// TwinCAT 3 PLC project cream_module_shell
// ProgramVersion: 3.1.0.8
// libraries:
//   Tc2_Standard, * (Beckhoff Automation GmbH)
//   Tc2_System, * (Beckhoff Automation GmbH)
//   Tc3_Interfaces, * (Beckhoff Automation GmbH)
//   Tc3_Module, * (Beckhoff Automation GmbH)
//   Tc2_MC2,3.3.8.0,Beckhoff Automation GmbH
//   Tc2_TcpIp,3.3.2.0,Beckhoff Automation GmbH
//   Tc2_Utilities,3.3.7.0,Beckhoff Automation GmbH
// project tree:
//   DUTs/InternalDataTypes/ eMainState.TcDUT, eSubState.TcDUT
//   DUTs/Server DUTs/ DUT_MODE.TcDUT, DUT_PARAMETER_INPUT.TcDUT, DUT_PARAMETER_OUTPUT.TcDUT, DUT_SERVER_MODULE_INTERFACE.TcDUT, DUT_SERVER_MODULE_INTERFACE_INPUT.TcDUT, DUT_SERVER_MODULE_INTERFACE_OUTPUT.TcDUT, DUT_SERVER_PARAMETERINPUTARRAY.TcDUT, DUT_SERVER_PARAMETEROUTPUTARRAY.TcDUT, DUT_SERVER_SKILLINPUTARRAY.TcDUT, DUT_SERVER_SKILLOUTPUTARRAY.TcDUT, DUT_SERVER_SKILL_INPUT.TcDUT, DUT_SERVER_SKILL_OUTPUT.TcDUT, DUT_SERVER_STATEVALUEARRAY.TcDUT, DUT_STATEVALUES.TcDUT
//   DUTs/SimulationInterface/ MNG_APPLICATION_INPUTS_32BIT.TcDUT, MNG_APPLICATION_OUTPUTS_32BIT.TcDUT, MNG_DataArray.TcDUT, MNG_DatagramHeader.TcDUT, MNG_DatagramType.TcDUT, MNG_POSE6.TcDUT, MNG_RawDatagram.TcDUT, MNG_TRAFO.TcDUT, VEC3.TcDUT
//   GVLs/ GVL.TcGVL, MI5.TcGVL, MNG_GLOBALS.TcGVL, OPCConstants.TcGVL
//   / PlcTask.TcTTO, SimuTask.TcTTO
//   POUs/ FB_EmergencyStop.TcPOU, FB_Error.TcPOU, FB_Init.TcPOU, FB_MoveAbs.TcPOU, FB_MoveRel.TcPOU, FB_Ready.TcPOU, FB_Refill.TcPOU, FB_ResetAxis.TcPOU, FB_ResetSystem.TcPOU, FB_StorageLevel.TcPOU, FB_Timer.TcPOU, FB_LogFifo.TcPOU, MAIN.TcPOU, MAIN_simu.TcPOU, MNG_SIMULATION.TcPOU, MNG_UPDATEIOS.TcPOU
// real-time tasks:
//   TASK PlcTask: cycle T#10ms, priority 20, ADS port 350
//   TASK SimuTask: cycle T#10ms, priority 21, ADS port 351
// motion (NC):
//   TASK NC-Task 1 SAF: cycle T#2ms, priority 4, ADS port 501
//   TASK NC-Task 1 SVB: cycle T#10ms, priority 8, ADS port 511
//   AXIS Axis 1 (id 1)
//     OtherSettings: AllowMotionCmdToSlave=true
//     encoder EncType=8
//       EncPara: MaxCount=#x0036ee7f
//     drive DrvType=9
//       DrvPara: MaxCount=#xffffffff, DriveControlDWord=#x00030000
//         Analog: VeloScale=6
//         TimeComp: TaskDelayCycles=1
//     controller CtrType=1
//       CtrPara: PriorControlFactor=1
//         Observer: BandWidth=20
// I/O:
//   DEVICE Device 1 (EtherCAT), AmsNetId 5.27.156.253.2.1
//     Term 1 (EK1200) [EK1200-5000 EtherCAT Power supply (2A E-Bus)]
//       Term 2 (EL1804) [EL1804 4Ch. Dig. Input 24V, 3ms]
//       Term 3 (EL3162) [EL3162 2Ch. Ana. Input 0-10V]
//       Term 4 (EK1110) [EK1110 EtherCAT extension]
//     Drive 5 (IndraDrive MPB16/17) [IndraDrive MPB16/17]
//   DEVICE Device 3 (RT-Ethernet Protocol), AmsNetId 5.27.156.253.4.1
//   DEVICE Device 2 (NOV-DP-RAM)
// variable links:
//   NC-Task 1 SAF/Axes/Axis 1 <-> Device 1 (EtherCAT)/Drive 5 (IndraDrive MPB16/17)
//     Drive/Inputs/In/nDcOutputTime <-> InfoData/DcOutputShift
//     Drive/Inputs/In/nState1 <-> AT/Drive status word @bit 8
//     Drive/Inputs/In/nState2 <-> AT/Drive status word
//     Drive/Inputs/In/nState4 @bit 1 <-> WcState/InputToggle
//     Drive/Inputs/In/nState4 <-> WcState/WcState
//     Drive/Outputs/Out/nCtrl1 <-> MDT/Master control word @bit 8
//     Drive/Outputs/Out/nDataOut1 <-> MDT/Position command value
//     Enc/Inputs/In/nDataIn1 <-> AT/Position feedback value 1
//     Enc/Inputs/In/nDcInputTime <-> InfoData/DcInputShift
//     Enc/Inputs/In/nState4 @bit 1 <-> WcState/InputToggle
//     Enc/Inputs/In/nState4 <-> WcState/WcState
//   cream_module_shell/cream_module_shell Instance <-> Device 1 (EtherCAT)/Term 1 (EK1200)/Term 2 (EL1804)
//     PlcTask Inputs/GVL.init_sensor <-> Channel 4/Input
//   cream_module_shell/cream_module_shell Instance <-> Device 1 (EtherCAT)/Term 1 (EK1200)/Term 3 (EL3162)
//     PlcTask Inputs/GVL.iPositionSens <-> AI Standard Channel 1/Value
//   cream_module_shell/cream_module_shell Instance <-> NC-Task 1 SAF/Axes/Axis 1
//     PlcTask Inputs/GVL.axis.NcToPlc <-> Outputs/ToPlc
//     PlcTask Outputs/GVL.axis.PlcToNc <-> Inputs/FromPlc

CONFIGURATION cream_module_shell
    RESOURCE PLC ON TwinCAT3
        TASK PlcTask(INTERVAL := T#10ms, PRIORITY := 20);
        TASK SimuTask(INTERVAL := T#10ms, PRIORITY := 21);
        PROGRAM MAIN WITH PlcTask : MAIN;
        PROGRAM MAIN_simu WITH SimuTask : MAIN_simu;
    END_RESOURCE
END_CONFIGURATION

// ---- DUTs/InternalDataTypes/eMainState.TcDUT
TYPE eMainState :
(
	init			:= 0,
	ready			:= 10,
	output			:= 20,
	empty			:= 30,
	refill			:= 40,
	emergencyStop	:= 50,
	error			:= 60,
	resetSystem		:= 70
);
END_TYPE

// ---- DUTs/InternalDataTypes/eSubState.TcDUT
TYPE eSubState :
(
	step0 := 0,
	step1 := 10,
	step2 := 20,
	step3 := 30,
	step4 := 40,
	step5 := 50,
	step6 := 60,
	step7 := 70,
	step8 := 80,
	step9 := 90,
	step10 := 100,
	step11 := 110,
	step12 := 120,
	step13 := 130,
	step14 := 140,
	step15 := 150
);
END_TYPE

// ---- DUTs/Server DUTs/DUT_MODE.TcDUT
/// MODE to run (inside of MODULE_INTERFACE_INPUT)
TYPE DUT_MODE :
(
	///Initialitzation number mode
	Init := 0,
	///Automatic number mode
	Auto := 1,
	///Manual number mode
	Manual := 2,
	Reset := 3
);
END_TYPE

// ---- DUTs/Server DUTs/DUT_PARAMETER_INPUT.TcDUT
TYPE DUT_PARAMETER_INPUT :
STRUCT
	///Value of the parameter 
	Value: LREAL;
	///Possibility to a string value depending on the parameter
	StringValue: STRING(80);
END_STRUCT
END_TYPE

// ---- DUTs/Server DUTs/DUT_PARAMETER_OUTPUT.TcDUT
TYPE DUT_PARAMETER_OUTPUT :
STRUCT
	///Free to use = TRUE, busy to use =FALSE
	Dummy: BOOL := TRUE;
	///ID of the parameter
	ID: UINT;
	///Name of the parameter
	Name: STRING(80);
	///Unit of the parameter
	Unit: STRING(80);
	///Optional parameter
	Required: BOOL;
	///Default parameter to work
	Default: LREAL;
	///Minimum value of the parameter
	MinValue: LREAL;
	///Maximum value of the parameter
	MaxValue: LREAL;
END_STRUCT
END_TYPE

// ---- DUTs/Server DUTs/DUT_SERVER_MODULE_INTERFACE.TcDUT
/// MODULE INTERFACE INPUT AND OUTPUT 
TYPE DUT_SERVER_MODULE_INTERFACE :
STRUCT
	///Information that the module reads
	Input: DUT_SERVER_MODULE_INTERFACE_INPUT;
	///Information that the module write
	Output: DUT_SERVER_MODULE_INTERFACE_OUTPUT;
END_STRUCT
END_TYPE

// ---- DUTs/Server DUTs/DUT_SERVER_MODULE_INTERFACE_INPUT.TcDUT
TYPE DUT_SERVER_MODULE_INTERFACE_INPUT :
STRUCT
	///Mode to run (init,auto,manual,..)
	Mode: INT;
	///check if the modules is alive
	ConnectionTestInput: BOOL;
	///Modules get their position
	PositionInput : LREAL;
	///Update data= TRUE, No updatedata=FALSE
	Watchbit: BOOL;
	///Emergency stop
	EmergencyStop: BOOL;
	///Range of INPUT skills
	SkillInput: DUT_SERVER_SKILLINPUTARRAY;
END_STRUCT
END_TYPE

// ---- DUTs/Server DUTs/DUT_SERVER_MODULE_INTERFACE_OUTPUT.TcDUT
TYPE DUT_SERVER_MODULE_INTERFACE_OUTPUT :
STRUCT
	///Free to use = TRUE, busy to use =FALSE
	Dummy: BOOL := TRUE;
	///Individual name of the module
	Name: STRING(80);
	///Identification number of module
	ID: UINT;
	///IP address
	IP: STRING(80);
	///Show if the module is in Standby or not
	Idle: BOOL;
	///Show if the module is connected
	Connected: BOOL;
	///Feedback with conection test input
	ConnectionTestOutput: BOOL;
	///Show if the system has error when=TRUE
	Error: BOOL;
	///Identification number of the error
	ErrorID: UINT;
	///Description of the error
	ErrorDescription: STRING(80);
	///Description of the current task
	CurrentTaskDescription: STRING(80);
	///Position of the output
	PositionOutput: LREAL;
	/// Bool value of the Sensor
	PositionSensor: BOOL;
	///Range of OUTPUT skills
	SkillOutput: DUT_SERVER_SKILLOUTPUTARRAY;
	///Range of state values
	StateValue: DUT_SERVER_STATEVALUEARRAY;
END_STRUCT
END_TYPE

// ---- DUTs/Server DUTs/DUT_SERVER_PARAMETERINPUTARRAY.TcDUT
TYPE DUT_SERVER_PARAMETERINPUTARRAY :
STRUCT
	ParameterInput0: DUT_PARAMETER_INPUT;
	ParameterInput1: DUT_PARAMETER_INPUT;
	ParameterInput2: DUT_PARAMETER_INPUT;
	ParameterInput3: DUT_PARAMETER_INPUT;
	ParameterInput4: DUT_PARAMETER_INPUT;
	ParameterInput5: DUT_PARAMETER_INPUT;
END_STRUCT
END_TYPE

// ---- DUTs/Server DUTs/DUT_SERVER_PARAMETEROUTPUTARRAY.TcDUT
TYPE DUT_SERVER_PARAMETEROUTPUTARRAY :
STRUCT
	ParameterOutput0: DUT_PARAMETER_OUTPUT;
	ParameterOutput1: DUT_PARAMETER_OUTPUT;
	ParameterOutput2: DUT_PARAMETER_OUTPUT;
	ParameterOutput3: DUT_PARAMETER_OUTPUT;
	ParameterOutput4: DUT_PARAMETER_OUTPUT;
	ParameterOutput5: DUT_PARAMETER_OUTPUT;
END_STRUCT
END_TYPE

// ---- DUTs/Server DUTs/DUT_SERVER_SKILLINPUTARRAY.TcDUT
TYPE DUT_SERVER_SKILLINPUTARRAY :
STRUCT
	SkillInput0: DUT_SERVER_SKILL_INPUT;
	SkillInput1: DUT_SERVER_SKILL_INPUT;
	SkillInput2: DUT_SERVER_SKILL_INPUT;
	SkillInput3: DUT_SERVER_SKILL_INPUT;
	SkillInput4: DUT_SERVER_SKILL_INPUT;
	SkillInput5: DUT_SERVER_SKILL_INPUT;
	SkillInput6: DUT_SERVER_SKILL_INPUT;
	SkillInput7: DUT_SERVER_SKILL_INPUT;
	SkillInput8: DUT_SERVER_SKILL_INPUT;
	SkillInput9: DUT_SERVER_SKILL_INPUT;
	SkillInput10: DUT_SERVER_SKILL_INPUT;
	SkillInput11: DUT_SERVER_SKILL_INPUT;
	SkillInput12: DUT_SERVER_SKILL_INPUT;
	SkillInput13: DUT_SERVER_SKILL_INPUT;
	SkillInput14: DUT_SERVER_SKILL_INPUT;
	SkillInput15: DUT_SERVER_SKILL_INPUT;
END_STRUCT
END_TYPE

// ---- DUTs/Server DUTs/DUT_SERVER_SKILLOUTPUTARRAY.TcDUT
TYPE DUT_SERVER_SKILLOUTPUTARRAY :
STRUCT
	SkillOutput0: DUT_SERVER_SKILL_OUTPUT;
	SkillOutput1: DUT_SERVER_SKILL_OUTPUT;
	SkillOutput2: DUT_SERVER_SKILL_OUTPUT;
	SkillOutput3: DUT_SERVER_SKILL_OUTPUT;
	SkillOutput4: DUT_SERVER_SKILL_OUTPUT;
	SkillOutput5: DUT_SERVER_SKILL_OUTPUT;
	SkillOutput6: DUT_SERVER_SKILL_OUTPUT;
	SkillOutput7: DUT_SERVER_SKILL_OUTPUT;
	SkillOutput8: DUT_SERVER_SKILL_OUTPUT;
	SkillOutput9: DUT_SERVER_SKILL_OUTPUT;
	SkillOutput10: DUT_SERVER_SKILL_OUTPUT;
	SkillOutput11: DUT_SERVER_SKILL_OUTPUT;
	SkillOutput12: DUT_SERVER_SKILL_OUTPUT;
	SkillOutput13: DUT_SERVER_SKILL_OUTPUT;
	SkillOutput14: DUT_SERVER_SKILL_OUTPUT;
	SkillOutput15: DUT_SERVER_SKILL_OUTPUT;
END_STRUCT
END_TYPE

// ---- DUTs/Server DUTs/DUT_SERVER_SKILL_INPUT.TcDUT
TYPE DUT_SERVER_SKILL_INPUT :
STRUCT
	///Range of parameters
	ParameterInput: DUT_SERVER_PARAMETERINPUTARRAY;
	///Start process
	Execute: BOOL;
END_STRUCT
END_TYPE

// ---- DUTs/Server DUTs/DUT_SERVER_SKILL_OUTPUT.TcDUT
TYPE DUT_SERVER_SKILL_OUTPUT :
STRUCT
	///Free to use = TRUE, busy to use =FALSE
	Dummy: BOOL := TRUE;
	///Identification number of skill
	ID: UINT;
	///indentfication name of skill
	Name: STRING(80);
	///Skill activated
	Activated: BOOL;
	///Ready to do skill
	Ready: BOOL;
	///Skill in process
	Busy: BOOL;
	///Skill finish
	Done: BOOL;
	///Error in system
	Error: BOOL;
	///Range of parameters
	ParameterOutput: DUT_SERVER_PARAMETEROUTPUTARRAY;
END_STRUCT
END_TYPE

// ---- DUTs/Server DUTs/DUT_SERVER_STATEVALUEARRAY.TcDUT
TYPE DUT_SERVER_STATEVALUEARRAY :
STRUCT
	StateValue0: DUT_STATEVALUES;
	StateValue1: DUT_STATEVALUES;
	StateValue2: DUT_STATEVALUES;
	StateValue3: DUT_STATEVALUES;
	StateValue4: DUT_STATEVALUES;
	StateValue5: DUT_STATEVALUES;
	StateValue6: DUT_STATEVALUES;
	StateValue7: DUT_STATEVALUES;
	StateValue8: DUT_STATEVALUES;
	StateValue9: DUT_STATEVALUES;
	StateValue10: DUT_STATEVALUES;
END_STRUCT
END_TYPE

// ---- DUTs/Server DUTs/DUT_STATEVALUES.TcDUT
TYPE DUT_STATEVALUES :
STRUCT
	///Free to use = TRUE, busy to use =FALSE
	Dummy: BOOL := TRUE;
	///Value of the State
	Value: LREAL;
	///Name of the state
	Name: STRING(80);
	///Description of the state
	Description: STRING(80);
	///Unit of the state ()
	Unit: STRING(80);
END_STRUCT
END_TYPE

// ---- DUTs/SimulationInterface/MNG_APPLICATION_INPUTS_32BIT.TcDUT

TYPE MNG_APPLICATION_INPUTS_32BIT :
STRUCT
    NumSignals                     : INT     := 5         ;
    HallSensor1_00_IR : BOOL    := 0; (* ysics/Keksmodul/Keksmodul - relevant/HallSensor1?IR *)
    HallSensor2_00_IR : BOOL    := 0; (* ysics/Keksmodul/Keksmodul - relevant/HallSensor2?IR *)
    init_sensor_cookie_module_00_IR : BOOL    := 0; (* l/Keksmodul - relevant/init_sensor_cookie_module?IR *)
    kein_cookie_mehr_00_IR : BOOL    := 0; (* /Keksmodul/Keksmodul - relevant/kein_cookie_mehr?IR *)
    cookiebox_sensor_00_IR : BOOL    := 0; (* Physics://physics/Keksmodul/cookiebox_sensor?IR *)
END_STRUCT
END_TYPE

// ---- DUTs/SimulationInterface/MNG_APPLICATION_OUTPUTS_32BIT.TcDUT

TYPE MNG_APPLICATION_OUTPUTS_32BIT :
STRUCT
    NumSignals                     : INT     := 3         ;
    Disc_00_ACT_POS : REAL    := 0.0; (* ysics/Keksmodul/Keksmodul - relevant/Disc?KinActual *)
    A2014_09_12_Left_Predeterminado_00_ACT_POS : REAL    := 0.0; (* nt/Scissor/2014_09_12_Left_Predeterminado?KinActual *)
    A2014_09_12_Right_Predeterminado_00_ACT_POS : REAL    := 0.0; (* t/Scissor/2014_09_12_Right_Predeterminado?KinActual *)
END_STRUCT
END_TYPE

// ---- DUTs/SimulationInterface/MNG_DataArray.TcDUT
TYPE MNG_DataArray : ARRAY[1..MNG_BUFFER_SIZE] OF DWORD; (* user data of max. length *)
END_TYPE

// ---- DUTs/SimulationInterface/MNG_DatagramHeader.TcDUT
TYPE MNG_DatagramHeader :(* datagram header (4 byte aligned) *)
STRUCT
	(* Time when datagram has been created *)
	Counter 	: DWORD;
	(* Time when datagram has been sent *)
	SentTime 		: DWORD;
	(* Type of the datagram *)
	DatagramType 	: DWORD := MNG_UnknownDatagram;
	(* Byte count in the payload *)
	ByteCount 		: DWORD := 0;
END_STRUCT
END_TYPE

// ---- DUTs/SimulationInterface/MNG_DatagramType.TcDUT
TYPE MNG_DatagramType :
(
	(*Dead man datagram signalizing peer is alive *)
	MNG_DeadManDatagram := 0,
	(*Time tick synchonisation *)
	MNG_TimeTick,
	(*Time tick synchonisation *)
	MNG_TimeTickRequest,
	(*Initialization of the connection *)
	MNG_InitConnection,
	(*Reset simulation *)
	MNG_ResetSimulation,
	(*Rewind simulation *)
	MNG_RewindSimulation,
	(*Start simulation *)
	MNG_StartSimulation,
	(*Stop simulation *)
	MNG_StopSimulation,
	(*IO Config datagram *)
	MNG_IOConfig,
	(*Complete Raw IO Image *)
	MNG_RawIOImage,
	(*Complete Raw 32 Bit IO Image *)
	MNG_Raw32BitImage,
	(*Delta IO, only ios that have changed *)
	(* IODelta, *)
	(*Text datagram *)
	MNG_TextDatagram,
	(*Unknown Datagram (future updates of peer, not supported by this side) *)
	MNG_UnknownDatagram
);
END_TYPE

// ---- DUTs/SimulationInterface/MNG_POSE6.TcDUT
TYPE MNG_POSE6 :(* position and orientation as an euler based pose *)
STRUCT
	x, y, z, a, b, c : REAL;
END_STRUCT
END_TYPE

// ---- DUTs/SimulationInterface/MNG_RawDatagram.TcDUT
TYPE MNG_RawDatagram :(* binary TCP/IP datagram (4 byte aligned) *)
STRUCT
	Header	:  MNG_DatagramHeader;(* datagram header *)
	Payload	:  MNG_DataARRAY;
END_STRUCT
END_TYPE

// ---- DUTs/SimulationInterface/MNG_TRAFO.TcDUT
TYPE MNG_TRAFO :(* position and orientation as a 4x4 matrix *)
STRUCT
	baseX : VEC3; 
	fill0 : REAL;
	baseY : VEC3; 
	fill1 : REAL;
	baseZ : VEC3; 
	fill2 : REAL;
	origin : VEC3;
	fill3 : REAL;
END_STRUCT
END_TYPE

// ---- DUTs/SimulationInterface/VEC3.TcDUT
TYPE VEC3 :(* 3d position *)
STRUCT
	x, y, z : REAL;
END_STRUCT
END_TYPE

// ---- GVLs/GVL.TcGVL
VAR_GLOBAL
	pi : REAL := 3.14159;
																
	//<<Input Variables>>//
	iPositionSens	AT%I*	: INT;			// Position of extruder from sensor
	
	//OPC input Variables
	creamType				: INT;			// chocolate = 0, strawberry jam = 1, apricot jam = 2, cheese = 3
	optionalExtraCream		: INT;			// plenty = 0, normal = 1
	
	//<<Output Variables>>//
	oModulePosition			: LREAL;
	
	//<<Internal Variables>>//
	axis	 				: AXIS_REF;
	
	mainState 				: eMainState	:= eMainState.init;
	emptySubState			: eSubState 	:= eSubState.step0;	
	refillSubState			: eSubState		:= eSubState.step0;
	initSubState			: eSubState		:= eSubstate.step0;
	readySubState			: eSubState		:= eSubstate.step0;
	emergencySubState		: eSubState		:= eSubstate.step0;
	errorSubState			: eSubState		:= eSubstate.step0;
	resetSubState			: eSubState		:= eSubstate.step0;
	
	modulePositionInitialized	: BOOL := FALSE;	// is the module position initialized?
	firstRun					: bool := true;		// is this the first init? then wait for axis to get ready
	
	iMotorPosition			: LREAL;		//Position of extruder from motor encoder
	
	stepWidth				: LREAL;					//step width for motor to get optimal cream amount
	stepBackWidth			: LREAL;					//step width for motor to get optimal cream amount
	slowVel					: LREAL			:= 2.0;		// velocity for pressing cream out
	fastVel					: LREAL			:= 20.0;	// velocity for going back to full position
	fullPos					: LREAL			:= 89.0;	// Position where extruder is full
	emptyPos				: LREAL			:= 0.0;		// Position where extruder is empty

	//<<For Simulation>>//
	offset					: LREAL;
	infinitsimu				: BOOL;
	infinitsimu2			: BOOL;
	init_sensor		AT%I*	: BOOL;
	SensorPosition			: LREAL;
	
END_VAR

// ---- GVLs/MI5.TcGVL
VAR_GLOBAL
	//<<OPC-UA Module Interface>>//
	{attribute 'OPC.UA.DA' := '1'}
	Module2301 : DUT_SERVER_MODULE_INTERFACE;
	{attribute 'OPC.UA.DA' := '1'}
	mySkillID : INT := 1230;		//default: 1230 raspberry jam, 1240 for apple sauce, 1250 for apricot
	{attribute 'OPC.UA.DA' := '1'}
	reset : BOOL := false;
END_VAR

// ---- GVLs/MNG_GLOBALS.TcGVL

VAR_GLOBAL CONSTANT
	PLCPRJ_MAX_CONNECTIONS					: UDINT 	:= 5;   (* Max. number of server<->client connections *)
	PLCPRJ_SERVER_RESPONSE_TIMEOUT			: TIME 	:= T#10s;
	PLCPRJ_CLIENT_SEND_CYCLE_TIME			: TIME 	:= T#1ms;

	PLCPRJ_RECEIVER_POLLING_CYCLE_TIME		: TIME 	:= T#1ms;
	PLCPRJ_BUFFER_SIZE						: UDINT	:= 10000;   (* Max. internal fifo/receiver buffer size *)

	(* Some project specific error codes *)
	PLCPRJ_ERROR_RECEIVE_BUFFER_OVERFLOW	: UDINT := 16#8101; (* receive fifo/buffer overflow*)
	PLCPRJ_ERROR_SEND_BUFFER_OVERFLOW		: UDINT := 16#8102;	(* send fifo/buffer overflow *)
	PLCPRJ_ERROR_RESPONSE_TIMEOUT			: UDINT := 16#8103;	(* receive timeout error *)
	
	

	PLCPRJ_ERROR_INVALID_FRAME_FORMAT		: UDINT := 16#8104;	(* invalid frame format/data *)
	PLCPRJ_ERROR_INVALID_IO_FORMAT_RECEIVED : UDINT := 16#8105;	(* invalid io format/data *)
	PLCPRJ_ERROR_INTERNAL					: UDINT := 16#8105; (* internal error *)
	PLCPRJ_ERROR_RX_DATA_INCONSISTENT		: UDINT := 16#8106; (* rx data inconsistent *)
	
	PLCPRJ_ERROR_RECEIVE_TIMEOUT			: UDINT := 16#8107;
	PLCPRJ_ERROR_SENDFIFO_OVERFLOW			: UDINT := 16#8108; (* send fifo overflow error *)
	PLCPRJ_ERROR_RECFIFO_OVERFLOW			: UDINT := 16#8109; (* receive fifo overflow error *)
	
    MNG_BUFFER_SIZE						: DWORD := 32768;   (* Bytes: 131072; Max 128 KB of datagram payload data*)
	MNG_DatagramsFIFO_Size					: DWORD := 10;      (* Max 10 datagrams buffered before loss occurs *)
	MNG_EmptyDatagramHeader					: MNG_DatagramHeader;
	MNG_Application_NumInputs				: DWORD := 4;
	MNG_Application_NumOutputs				: DWORD := 4;

        (* PI should be defined by the system *)
        (* PI      : LREAL := 3.1415926535897932384626433832795; *)
        DEG2RAD : LREAL := 0.017453292519943295769236907684886;
        RAD2DEG : LREAL := 57.295779513082320876798154814105;
END_VAR

VAR_GLOBAL
        MNG_TIMESTAMP                                           : LREAL := 0;
END_VAR

// ---- GVLs/OPCConstants.TcGVL
VAR_GLOBAL CONSTANT
	///Maximum number of skillparameters
	ParameterCnt: INT := 5;
	///Maximum number of skills per Module
	SkillCnt: INT := 15;
	///Maximum number of Statevalues of one Module
	StateCnt: INT := 10;
	///Maximum number of modules
	ModuleCnt: INT := 10;
	///Maximum number of Tasks in Production List
	TaskCnt: INT := 30;
	///Maximum number  of offered recipes
	OfferCnt: INT := 5;
	///Maximum number of Orders in Queue
	OrderCnt: INT := 5;
	///Number of user set parameters per recipe
	UserParameterCnt: INT := 5;
	///Number of skills per task
	TaskSkillCnt: INT := 50;
END_VAR

// ---- POUs/MAIN.TcPOU
PROGRAM MAIN
VAR
	FBI_init			: FB_Init;			//FBI = function block instance
	FBI_refill			: FB_Refill;
	FBI_ready			: FB_Ready;
	FBI_emergencyStop 	: FB_EmergencyStop;
	FBI_error 			: FB_Error;
	FBI_storageLevel	: FB_StorageLevel;
	FBI_resetSystem		: FB_ResetSystem;  

	
	//jonas Interface variables:
	FBI_Timer			: TOF;
END_VAR

// @TODO measure position of slide against position sensor of XTS

//----------------------------------------- Error handling and emergency stop ------------------------------------------
axis.ReadStatus();

//reset system
IF (MI5.reset) THEN	
	GVL.mainState := eMainState.resetSystem;

//Emergency Stop Watchdog!	
ELSIF Module2301.Input.EmergencyStop THEN		
	GVL.mainState := eMainState.emergencyStop;

// error handling
ELSIF (axis.Status.Error) THEN					
	GVL.mainState := eMainState.error;
	
END_IF


//------------------------------------------------ OPC UA and module init --------------------------------------------------------------

//Connection Test
Module2301.Output.ConnectionTestOutput := Module2301.Input.ConnectionTestInput;
//positionsweitergabe an procvess tool
Module2301.Output.PositionOutput := Module2301.Input.PositionInput + 31;

//module positioning (by jf)
FBI_Timer();
IF GVL.init_sensor THEN
	Module2301.Output.PositionSensor := TRUE;
	FBI_Timer(IN := TRUE,PT := T#400MS);
	FBI_Timer(IN := FALSE,PT := T#400MS);
ELSE
	Module2301.Output.PositionSensor := FBI_Timer.Q;
END_IF


//----------------------------------------------- cream function process and parameter reading ----------------------------------------------------

// determine stepWidth from creamType
IF (MI5.mySkillID = 1230 OR MI5.mySkillID = 1250) THEN				// raspberry jam or apricot
	GVL.stepWidth := -3.5 - (Module2301.Input.SkillInput.SkillInput0.ParameterInput.ParameterInput0.Value / 100);
	GVL.stepBackWidth := 2;
ELSIF (MI5.mySkillID = 1240) THEN			// applesauce
	GVL.stepWidth := -4.5 - (Module2301.Input.SkillInput.SkillInput0.ParameterInput.ParameterInput0.Value / 100);
	GVL.stepBackWidth := 3;
END_IF


// get constantly the position of extruder
GVL.iMotorPosition := axis.NcToPlc.ActPos;

// update motor position for simulation
Module2301.Output.StateValue.StateValue2.Value := GVL.iMotorPosition;

//calculate storage level
FBI_storageLevel();


//----------------------------------------------- pseudo function block calls ----------------------------------------------------------------------

CASE GVL.mainState OF

	eMainState.init: //<<<<<<<<<<<<<<<<<<<<<<<<<<<<<<<<<<<<<<<<<<<<<<<<<<<<<<<<<<<<<<
		//init of state whereever the position of the disk is
		FBI_init();
	
	eMainState.ready: //<<<<<<<<<<<<<<<<<<<<<<<<<<<<<<<<<<<<<<<<<<<<<<<<<<<<<<<<<<<<<
		//cookie is on the clamps, waiting for putting it on the mover
		FBI_ready();
	
	eMainState.refill: //<<<<<<<<<<<<<<<<<<<<<<<<<<<<<<<<<<<<<<<<<<<<<<<<<<<<<<<<<<<<
		//cookie storage empty --> needs to be refilled
		FBI_refill();
		
	eMainState.emergencyStop: //<<<<<<<<<<<<<<<<<<<<<<<<<<<<<<<<<<<<<<<<<<<<<<<<<<<<<<<<<<<<
		// manually set emergency stop
		FBI_emergencyStop();
		
	eMainState.error: //<<<<<<<<<<<<<<<<<<<<<<<<<<<<<<<<<<<<<<<<<<<<<<<<<<<<<<<<<<<<
		// error state
		FBI_error();
		
	eMainState.resetSystem: //<<<<<<<<<<<<<<<<<<<<<<<<<<<<<<<<<<<<<<<<<<<<<<<<<<<<<<<<<<<<
		//error state
		FBI_resetSystem(); 
		
END_CASE

END_PROGRAM

// ---- POUs/FB_Init.TcPOU
FUNCTION_BLOCK FB_Init
VAR_INPUT
END_VAR
VAR_OUTPUT	
END_VAR
VAR
	resetAxis	: FB_ResetAxis;
	timer		: FB_Timer;
END_VAR

//@TODO: Determine the correct difference between sensor value and motorposition

//>>>OPCUA Init<<<
CASE initSubState OF	
			
step0:		// wait for everything to boot in first run
			IF (firstRun) THEN
				timer(iTime:=T#5S, execute := TRUE);
				IF(timer.done) THEN
					firstRun := FALSE;
				END_IF
			ELSE
				initSubState := step1;
			END_IF

step1:		//reset all substates
			emptySubState := step0;
			refillSubState := step0;
			readySubState := step0;
			emergencySubState := step0;
			errorSubState := step0;

			//>>>OPCUA Init<<<
			//>Module<
			Module2301.Output.ID := 2301;
			Module2301.Output.Name := 'Cream module Beckhoff';
			Module2301.Output.IP := '192.168.192.138';
			Module2301.Output.CurrentTaskDescription := 'Init process started: OPC UA';
			Module2301.Output.Dummy := FALSE;
			Module2301.Output.Idle := FALSE;
			Module2301.Output.Error := FALSE;
			Module2301.Output.ErrorDescription := '';
			Module2301.Output.ErrorID := 0;			
			
			//>Skill<:
			//Skill Cream
			Module2301.Output.SkillOutput.SkillOutput0.ID := mySkillID;
			Module2301.Output.SkillOutput.SkillOutput0.Activated := TRUE;
			Module2301.Output.SkillOutput.SkillOutput0.Busy := TRUE;
			Module2301.Output.SkillOutput.SkillOutput0.Done := FALSE;
			Module2301.Output.SkillOutput.SkillOutput0.Error := FALSE;
			Module2301.Output.SkillOutput.SkillOutput0.Ready := FALSE;
			Module2301.Output.SkillOutput.SkillOutput0.Dummy := FALSE;
			
			// publish maximum level of cream for HMI
			Module2301.Output.StateValue.StateValue1.Description := 'Maximum level of cream in injection.';
			Module2301.Output.StateValue.StateValue1.Dummy := FALSE;
			Module2301.Output.StateValue.StateValue1.Name := 'Max. Cream';
			Module2301.Output.StateValue.StateValue1.Unit := 'ml';
			Module2301.Output.StateValue.StateValue1.Value := 113;
			
			// publish motor position for simulation
			Module2301.Output.StateValue.StateValue2.Description := 'Motor Position.';
			Module2301.Output.StateValue.StateValue2.Dummy := FALSE;
			Module2301.Output.StateValue.StateValue2.Name := 'Motor Position';
			Module2301.Output.StateValue.StateValue2.Unit := 'mm';
			
			//initialize position input with value -1
			IF (NOT GVL.modulePositionInitialized)THEN
				Module2301.Input.PositionInput := -1;
				GVL.modulePositionInitialized := TRUE;
			END_IF
							
			resetAxis (execute := FALSE);
			
			IF (axis.Status.StandStill OR axis.Status.ErrorStop OR axis.Status.Disabled) THEN
				initSubState := step2;
			END_IF			

			
step2:		IF NOT resetAxis.done THEN
				// axreset
				resetAxis (execute := TRUE);
			ELSE
				initSubState := step3;
			END_IF
			
			
step3:		IF (iMotorPosition <=5) THEN
				mainState := eMainState.refill;
			ELSE
				mainState := eMainState.ready;
			END_IF
				initSubState := step0;
END_CASE

END_FUNCTION_BLOCK

// ---- POUs/FB_ResetAxis.TcPOU
FUNCTION_BLOCK FB_ResetAxis
VAR_INPUT
	execute: BOOL;
END_VAR
VAR_OUTPUT
	done : BOOL;
	busy : BOOL;
	error: BOOL;
END_VAR
VAR
	state			: INT := 0;
	fbreset			: Tc2_MC2.MC_Reset;
END_VAR

IF execute THEN
	CASE state OF
	
	0: 
		done := FALSE;
		fbreset(axis := axis, Execute := FALSE);
		state := 1;
		
	1:
		fbreset(
				Axis:= axis, 
				Execute:= TRUE, 
				Done=> , 
				Busy=> , 
				Error=> error, 
				ErrorID=> );
		IF fbreset.Done THEN
			state := 2;
		END_IF
		
	2:	
		execute := FALSE;
		done  := TRUE;
		state := 0;

	END_CASE
ELSE
	done := FALSE;
	state := 0;
END_IF

END_FUNCTION_BLOCK

// ---- POUs/FB_Timer.TcPOU
FUNCTION_BLOCK FB_Timer
VAR_INPUT
	iTime	: TIME;
	execute : Bool;
END_VAR
VAR_OUTPUT
	done	: BOOL;
END_VAR
VAR
	timer	: Tc2_Standard.TON;
	state	: INT := 0;
END_VAR

IF (execute) THEN
	
	CASE state OF
	
		0:	done := FALSE;
			timer(IN:= FALSE, PT:= iTime);
			timer(IN:= TRUE, PT:= iTime);
			state := 10;
	
		10:	timer();
			IF (timer.Q) THEN
				done := TRUE;
				state :=0;
			END_IF
	END_CASE

ELSE
	state := 0;
	done := FALSE;
END_IF

END_FUNCTION_BLOCK

// ---- POUs/FB_Refill.TcPOU
FUNCTION_BLOCK FB_Refill
VAR_INPUT
END_VAR
VAR_OUTPUT
END_VAR
VAR
	moveAbs : FB_MoveAbs;
END_VAR

CASE refillSubState OF

	step0:	//set OPC state variables
			Module2301.Output.SkillOutput.SkillOutput0.Busy := TRUE;
			Module2301.Output.SkillOutput.SkillOutput0.Done := FALSE;
			Module2301.Output.SkillOutput.SkillOutput0.Error := FALSE;
			Module2301.Output.SkillOutput.SkillOutput0.Ready := FALSE;
			
			//reset move functions
			moveAbs(execute := FALSE);
			
			refillSubState := step1; 
	
	step1:	//Move back to position with cream extruder beeing fully extended
			moveAbs(targetPos:= GVL.fullPos, targetVel:= GVL.fastVel, execute:= TRUE);
			IF (moveAbs.done) THEN
				refillSubState := step2; 
			END_IF
			

	step2:	//go in the right error state
			Module2301.Output.SkillOutput.SkillOutput0.Busy := FALSE;
			Module2301.Output.CurrentTaskDescription := 'Cream empty. Switching to refill mode.';
			Module2301.Output.ErrorID := 201;
			Module2301.Output.Error := TRUE;
			Module2301.Output.ErrorDescription := 'storage empty. please refill';
			refillSubState := step3;
			
	step3:	//wait for process tool to set the module in manual mode
			IF(Module2301.Input.Mode = DUT_MODE.Manual) THEN
				refillSubState := step4;
			END_IF
			
	step4:	//wait for process tool to set the module in init mode
			IF(Module2301.Input.Mode = DUT_MODE.Auto) THEN
				//reset error 
				Module2301.Output.Error := FALSE;
				Module2301.Output.ErrorDescription := '';
				Module2301.Output.ErrorID := 0;
				
				//change to ready state
				mainState := eMainState.ready;
				refillSubState := step0;
			END_IF
END_CASE

END_FUNCTION_BLOCK

// ---- POUs/FB_MoveAbs.TcPOU
FUNCTION_BLOCK FB_MoveAbs
VAR_INPUT
	targetPos		: LREAL;
	targetVel		: LREAL;
	execute			: BOOL := TRUE;
	
END_VAR

VAR_OUTPUT
	done 			: BOOL;
	moveAbs			: Tc2_MC2.MC_MoveAbsolute;
END_VAR

VAR
	state		: INT := -10;
	power		: Tc2_MC2.MC_Power;
END_VAR

//Comment here
IF (NOT execute) THEN
	state := -10;
	moveAbs	(Axis:= axis , Execute:= FALSE);
ELSE
	//Comment here
	power(
			Axis			:= axis , 
			Enable			:= TRUE , 
			Enable_Positive	:= TRUE , 
			Enable_Negative	:= TRUE , 
			BufferMode		:= Tc2_MC2.MC_BlendingNext
		);				
					
	CASE state OF 
		 
		-10:	//Comment here
				done := FALSE;
				IF (power.Status=TRUE AND power.Error=FALSE) THEN
					state := 0;
				END_IF
							
		0:		//Comment here
				moveAbs(Axis:= axis , Execute:= FALSE);
				state := 10;			
				
		10:		//Comment here
				IF (moveAbs.Done=FALSE) THEN
					moveAbs(Axis:= axis, Execute:= TRUE, Position:= targetPos, Velocity:=targetVel, BufferMode:= Tc2_MC2.MC_BlendingNext);
				ELSE 
					moveAbs(Axis:= axis, Execute:= FALSE);
					state := 20;
				END_IF
				
		20: 	//Comment here
				done 	:= TRUE;
				execute := false;
				state	:= -10;	
	END_CASE
END_IF

END_FUNCTION_BLOCK

// ---- POUs/FB_Ready.TcPOU
FUNCTION_BLOCK FB_Ready
VAR_INPUT
END_VAR
VAR_OUTPUT
END_VAR
VAR
	moveRel : FB_MoveRel;
END_VAR

CASE readySubState OF

step0:	moveRel(execute := false);
		IF (NOT (Module2301.Input.PositionInput = -1)) THEN
			readySubState := step1;
		END_IF

step1:	Module2301.Output.SkillOutput.SkillOutput0.Busy := FALSE;
		Module2301.Output.SkillOutput.SkillOutput0.Done := FALSE;
		Module2301.Output.SkillOutput.SkillOutput0.Error := FALSE;
		Module2301.Output.SkillOutput.SkillOutput0.Ready := TRUE;
		
		//wait for execute command
		IF(Module2301.Input.SkillInput.SkillInput0.Execute) THEN
		//order received
			Module2301.Output.SkillOutput.SkillOutput0.Ready := FALSE;
			Module2301.Output.SkillOutput.SkillOutput0.Busy := TRUE;
			readySubState := step2;
		END_IF
		
step2:	//@TODO: How much has the Bosch motor got to move to eject sufficient amount of cream?
		moveRel(targetDis:= GVL.stepWidth, targetVel:= GVL.slowVel, execute:= TRUE);
		IF (moveRel.done) THEN
			readySubState := step3; 
		END_IF
		
step3:	//@TODO: How much has the Bosch motor got to move to eject sufficient amount of cream?
		moveRel(targetDis:= GVL.stepBackWidth, targetVel:= GVL.slowVel, execute:= TRUE);
		IF (moveRel.done) THEN
			Module2301.Output.SkillOutput.SkillOutput0.Busy := FALSE;
			Module2301.Output.SkillOutput.SkillOutput0.Done := TRUE;
			readySubState := step4; 
		END_IF
		
step4:	// Test if distance sensor checks a position where the cream dispenser has to be empty
		IF (NOT Module2301.Input.SkillInput.SkillInput0.Execute) THEN
			IF (iMotorPosition <=5) THEN
				mainState := eMainState.refill;
			ELSE
				readySubState := step0;
			END_IF
		END_IF

END_CASE

END_FUNCTION_BLOCK

// ---- POUs/FB_MoveRel.TcPOU
FUNCTION_BLOCK FB_MoveRel
VAR_INPUT
	targetDis		: LREAL;
	targetVel		: LREAL;
	execute			: BOOL := TRUE;
	
END_VAR

VAR_OUTPUT
	done 			: BOOL;
	moveRel			: Tc2_MC2.MC_MoveRelative;
END_VAR

VAR
	state		: INT := -10;
	power		: Tc2_MC2.MC_Power;
END_VAR

//Comment here
IF (NOT execute) THEN
	state := -10;
	moveRel	(Axis:= axis , Execute:= FALSE);
ELSE
	//Comment here
	power(
			Axis			:= axis , 
			Enable			:= TRUE , 
			Enable_Positive	:= TRUE , 
			Enable_Negative	:= TRUE , 
			BufferMode		:= Tc2_MC2.MC_BlendingNext
		);				
					
	CASE state OF 
		 
		-10:	//Comment here
				done := FALSE;
				IF (power.Status=TRUE AND power.Error=FALSE) THEN
					state := 0;
				END_IF
							
		0:		//Comment here
				moveRel(Axis:= axis , Execute:= FALSE);
				state := 10;			
				
		10:		//Comment here
				IF (moveRel.Done=FALSE) THEN
					moveRel(Axis:= axis, Execute:= TRUE, Distance:= targetDis, Velocity:=targetVel, BufferMode:= Tc2_MC2.MC_BlendingNext);
				ELSE 
					moveRel(Axis:= axis, Execute:= FALSE);
					state := 20;
				END_IF
				
		20: 	//Comment here
				done 	:= TRUE;
				execute := false;
				state	:= -10;	
	END_CASE
END_IF

END_FUNCTION_BLOCK

// ---- POUs/FB_EmergencyStop.TcPOU
FUNCTION_BLOCK FB_EmergencyStop
VAR_INPUT
END_VAR
VAR_OUTPUT
END_VAR
VAR
END_VAR

CASE emergencySubState OF

	step0:	Module2301.Output.SkillOutput.SkillOutput0.Busy := FALSE;
			Module2301.Output.SkillOutput.SkillOutput0.Done := FALSE;
			Module2301.Output.SkillOutput.SkillOutput0.Dummy := FALSE;
			Module2301.Output.SkillOutput.SkillOutput0.Error := TRUE;
			Module2301.Output.SkillOutput.SkillOutput0.Ready := FALSE;
			
			//change in the right error state
			Module2301.Output.ErrorID := 302;
			Module2301.Output.CurrentTaskDescription := 'Emergency stop';
			Module2301.Output.Error := TRUE;
			Module2301.Output.ErrorDescription := 'Emergency stop. please solve problem';
			
			//wait for process tool to set the module in manual mode
			IF(Module2301.Input.Mode = DUT_MODE.Manual) THEN
				emergencySubState := step1;
			END_IF
			
	step1:	//wait for process tool to set the module in init mode
			IF(Module2301.Input.Mode = DUT_MODE.Auto) THEN
				//reset error 
				Module2301.Output.Error := FALSE;
				Module2301.Output.ErrorDescription := '';
				Module2301.Output.ErrorID := 0;

				//change to init state
				initSubState := step0;
				mainState := eMainState.init;
				emergencySubState := step0;
			END_IF
END_CASE

END_FUNCTION_BLOCK

// ---- POUs/FB_Error.TcPOU
FUNCTION_BLOCK FB_Error
VAR_INPUT
END_VAR
VAR_OUTPUT
END_VAR
VAR
	resetAxis			: FB_ResetAxis;
END_VAR

//@TODO: implement all possible errors

CASE errorSubState OF

	step0:	Module2301.Output.SkillOutput.SkillOutput0.Busy := FALSE;
			Module2301.Output.SkillOutput.SkillOutput0.Done := FALSE;
			Module2301.Output.SkillOutput.SkillOutput0.Dummy := FALSE;
			Module2301.Output.SkillOutput.SkillOutput0.Error := TRUE;
			Module2301.Output.SkillOutput.SkillOutput0.Ready := FALSE;
			
			// Error: axis got stuck
			IF (axis.Status.ErrorID = 17744) THEN
				Module2301.Output.ErrorDescription := 'Axis got stuck. Please clear module.';
				Module2301.Output.ErrorID := 301;
				errorSubState := step1;
			END_IF
			
			IF (Module2301.Output.ErrorID = 0) THEN
				Module2301.Output.ErrorDescription := 'Unknown Error.';
				Module2301.Output.ErrorID := 399;
				errorSubState := step1;
			END_IF
			
			//change in the right error state
			Module2301.Output.CurrentTaskDescription := 'Axis Error';
			Module2301.Output.Error := TRUE;
			
	step1:	//wait for process tool to set the module in manual mode
			IF(Module2301.Input.Mode = DUT_MODE.Manual) THEN
				resetAxis(execute:= FALSE);
				errorSubState := step2;
			END_IF
			
	step2:	IF NOT resetAxis.done THEN
				// axreset
				resetAxis (execute := TRUE);
			ELSE			
				errorSubState := step3;
			END_IF
			
	step3:	//wait for process tool to set the module in init mode
			IF(Module2301.Input.Mode = DUT_MODE.Auto) THEN
				//reset error 
				Module2301.Output.Error := FALSE;
				Module2301.Output.ErrorDescription := '';
				Module2301.Output.ErrorID := 0;
				
				//change to init state
				initSubState := step0;
				errorSubState := step0;
				mainState := eMainState.init;				
			END_IF
END_CASE

END_FUNCTION_BLOCK

// ---- POUs/FB_StorageLevel.TcPOU
FUNCTION_BLOCK FB_StorageLevel
VAR_INPUT
END_VAR
VAR_OUTPUT
END_VAR
VAR
	calculatedCream		: LREAL;
	remainingCream		: LREAL;		// in ml, is calculated by motor position
END_VAR

//Comment here	
IF (GVL.iPositionSens > 11090) THEN
	remainingCream := 0;
// configuration for all cookies (not as acurate)
ELSE
	calculatedCream := (11110 - GVL.iPositionSens)/86;
	remainingCream := REAL_TO_INT(calculatedCream);
END_IF

Module2301.Output.StateValue.StateValue0.Description := 'Remaining cream in the module.';
Module2301.Output.StateValue.StateValue0.Dummy := FALSE;
Module2301.Output.StateValue.StateValue0.Name := 'Remaining Cream';
Module2301.Output.StateValue.StateValue0.Unit := 'ml';
Module2301.Output.StateValue.StateValue0.Value := remainingCream;

END_FUNCTION_BLOCK

// ---- POUs/FB_ResetSystem.TcPOU
FUNCTION_BLOCK FB_ResetSystem
VAR_INPUT
END_VAR
VAR_OUTPUT
END_VAR
VAR
	resetAxis : FB_ResetAxis;
END_VAR

CASE GVL.resetSubState OF

step0:	resetAxis (execute := FALSE);

		Module2301.Output.SkillOutput.SkillOutput0.Busy := TRUE;
		Module2301.Output.SkillOutput.SkillOutput0.Done := TRUE;
		Module2301.Output.SkillOutput.SkillOutput0.Error := TRUE;
		Module2301.Output.SkillOutput.SkillOutput0.Ready := TRUE;
		
		GVL.resetSubState := step1;
		
step1:	IF NOT resetAxis.done THEN
		// axreset
		resetAxis (execute := TRUE);
		ELSE
			GVL.resetSubState := step2;
		END_IF
		
step2:	// reset substates
		GVL.emptySubState := step0;
		GVL.refillSubState := step0;
		GVL.initSubState := step0;
		GVL.readySubState := step0;
		GVL.emergencySubState := step0;
		GVL.errorSubState := step0;
		GVL.resetSubState := step0;
		
		MI5.reset := FALSE;
		GVL.mainState := eMainState.init;		
		
END_CASE

END_FUNCTION_BLOCK

// ---- POUs/MAIN_simu.TcPOU
PROGRAM MAIN_simu
VAR
    simIO 		: MNG_Simulation;
	outputs    	: MNG_Application_Outputs_32Bit;
    inputs     	: MNG_Application_Inputs_32Bit;
    ioUpdater  	: MNG_UpdateIOs                	:= (sRemoteHost := '192.168.175.222', nRemotePort := 5110);
	a 			: LREAL							:= 5.00;
    bEnable   	: BOOL                         	:= TRUE;
END_VAR

// Update IOs with simulation
//simIO(bEnable := TRUE);

// Application code follows here:
(*
IF GVL.infinitsimu THEN
	outputs.Disc_00_ACT_POS := (REAL_TO_INT(GVL.SensorPosition -180 + GVL.axis.NcToPlc.ModuloActPos))MOD 360;
ELSE
	IF GVL.infinitsimu2 THEN
		outputs.Disc_00_ACT_POS := (REAL_TO_INT(GVL.SensorPosition + GVL.axis.NcToPlc.ModuloActPos))MOD 360;
	ELSE
		outputs.Disc_00_ACT_POS := GVL.axis.NcToPlc.ModuloActPos;
	END_IF	
END_IF

storageLevel.full := inputs.kein_cookie_mehr_00_IR;

outputs.A2014_09_12_Right_Predeterminado_00_ACT_POS := ABS(SIN(((GVL.axis.NcToPlc.ActPos*pi)/180)))*(-7);
outputs.A2014_09_12_Left_Predeterminado_00_ACT_POS := ABS(SIN(((GVL.axis.NcToPlc.ActPos*pi)/180)))*(7);

GVL.iCookieInOutput := inputs.cookiebox_sensor_00_IR;
GVL.iDiskAtStorage := inputs.HallSensor1_00_IR;
GVL.iDiskAtRamp := inputs.HallSensor2_00_IR;

GVL.init_sensor := inputs.init_sensor_cookie_module_00_IR;

ioUpdater(Outputs := outputs, Inputs => inputs, bEnable := bEnable); 
*)
//outputs.Keksquelle_00_ReleaseTime := 60;
//outputs.Keksquelle_00_AlwaysOn := TRUE;

END_PROGRAM

// ---- POUs/MNG_SIMULATION.TcPOU
FUNCTION_BLOCK MNG_Simulation
VAR_INPUT
    bEnable    : BOOL                          := FALSE;
    outputs    : MNG_Application_Outputs_32Bit         ;
END_VAR
VAR_OUTPUT
    inputs     : MNG_Application_Inputs_32Bit          ;
END_VAR
VAR
    ioUpdater  : MNG_UpdateIOs                 := (sRemoteHost := '192.168.175.222', nRemotePort := 5110);
    fbCloseAll : FB_SocketCloseAll;
    bCloseAll  : BOOL := TRUE;
END_VAR

(* @END_DECLARATION := '0'                                                    *)
IF bCloseAll THEN (*On PLC reset or program download close all old (opened) connections *)
    bCloseAll := FALSE;
    fbCloseAll( bExecute:= TRUE );
ELSE
    fbCloseAll( bExecute:= FALSE );
END_IF

IF NOT fbCloseAll.bBusy THEN

    (* ------------------------------------- trigger data exchange ----------------------------------------------------------------------------*)
    ioUpdater(Outputs := outputs, Inputs => inputs, bEnable := bEnable);

END_IF

END_FUNCTION_BLOCK

// ---- POUs/MNG_UPDATEIOS.TcPOU
FUNCTION_BLOCK MNG_UpdateIOs
(* This function block implements simple TCP/IP client protocol.              *)
(* The max. size of binary tx/rx data has to be <= PLCPRJ_BUFFER_SIZE         *)
VAR_IN_OUT
    Outputs : MNG_Application_Outputs_32Bit;    (* Tx user data *)
END_VAR

VAR_INPUT
    bDbg        : BOOL                         := FALSE               ; (* TRUE => Enable debug output, FALSE => Disable debug output *)
    sRemoteHost : STRING(15)                   := '127.0.0.1'         ; (* IP address of remote server *)	
    nRemotePort : UDINT                        := 5000                ; (* Remote server port *)
    bEnable     : BOOL                         := FALSE               ; (* TRUE => Enable/connect, FALSE => Disable/disconnect *)
    tReconnect  : TIME                         := T#5s                ;
END_VAR

VAR_OUTPUT
    errors      : FB_LogFifo                                          ; (* Error message fifo *)
    Inputs      : MNG_Application_Inputs_32Bit                        ; (* Rx user data *)
    eState      : E_SocketConnectionState      := eSOCKET_DISCONNECTED; (* TCP/IP connection state *)
END_VAR

VAR
    counter          : DWORD                        := 0                   ;
    fbConnect        : FB_ClientServerConnection    := (tReconnect := T#5s); (* Create/release TCP/IP connection *)
    fbSend           : FB_SocketSend                                       ; (* Send TCP/IP data *)
    fbReceive        : FB_SocketReceive                                    ; (* Receive TCP/IP data *)
    state            : BYTE                                                ; (* Global state *)
    tx_state         : BYTE                                                ; (* Tx state *)
    rx_state         : BYTE                                                ; (* Rx state *)

    toServer         : MNG_RawDatagram                                     ;
    fromServer       : MNG_RawDatagram                                     ;
    cbReceived       : UDINT                                               ; (* Count of received data bytes *)
    cbRx             : UDINT                                               ; (* Rx frame byte size *)

    bDisconnect      : BOOL                                                ; (* Disconnect flag, if set the socket will be closed *)
    pollTimer        : TON                                                 ; (* Rx data poll timer *)
    bAbort           : BOOL                                                ; (* Flag to abort frame parsing loop *)
    sID              : STRING(20)                   := ''                  ;
    clock            : FB_LocalSystemTime           := ( bEnable := TRUE ) ; (* OS clock *)
    _byteCount       : DWORD                                               ;
    _i               : DWORD                                               ;
    _ptr             : POINTER TO BYTE                                     ;
    _internalInputs  : MNG_Application_Inputs_32Bit                        ;
    DWordBuffer      : DWORD                                               ; (* convert DWORD data *)
    DIntBuffer       : DINT                                                ; (* convert DINT data *)
END_VAR


(* refresh clock time                                                         *)
clock();

(* state chart                                                                *)
CASE state OF
    0:(* Init state *)
        (*rx.A_Reset(bDbg := bDbg)  ; (* Reset RX fifo (optional) *)
        tx.A_Reset    (bDbg := bDbg); (* Reset TX fifo (optional) *)*)
        errors.Clear(); (* Reset error fifo (optional) *)

        pollTimer( IN := FALSE, PT := PLCPRJ_RECEIVER_POLLING_CYCLE_TIME );
        bDisconnect := FALSE;(* Reset disconnect flag *)
        cbReceived  := 0;(* Reset number of received data bytes *)
        tx_state    := 0;(* Reset tx state machine *)
        rx_state    := 0;(* Reset rx state machine *)
        state       := 1;(* Go to the next step *)

    1:(* Create TCP/IP connection *)
        fbConnect(sSrvNetID := '',
                  nMode := CONNECT_MODE_ENABLEDBG,(* Enable debug output *)
                  sRemoteHost := sRemoteHost,
                  nRemotePort := nRemotePort,
                  tReconnect  := tReconnect,
                  bEnable     := bEnable,
                  eState      => eState);
        IF NOT fbConnect.bBusy THEN

            (* Create identification string used by debug messages *)
            sID          := CONCAT(CONCAT('[', DWORD_TO_HEXSTR(fbConnect.hSocket.handle, 4, FALSE) ), ']');
            errors.sMessage := CONCAT('CLI.Err', sID);

            IF NOT fbConnect.bError THEN
                IF eState = eSOCKET_CONNECTED THEN(* we are connected *)
                    state := 2;
                END_IF
            ELSE(* connect error: log error *)
                errors.Error(nErrId := fbConnect.nErrId);
            END_IF
        END_IF

    2:(* Data exchange state *)
        bDisconnect := NOT bEnable OR bDisconnect; (* user/internal disconnect requested? *)
        IF bDisconnect AND (tx_state = 0) AND (rx_state = 0) THEN
            state := 3;(* disconnect *)
        ELSE
            (*--------------------------- Send tx data -------------------------------------------*)
            CASE tx_state OF
                0:
                    IF NOT bDisconnect THEN

                        (* forcefully send data each cycle *)

                        (* create the raw datagram *)
                        _byteCount                   := 16;
                        toServer.Header.ByteCount    := HOST_TO_BE32(in := _byteCount);
                        toServer.Header.DatagramType := HOST_TO_BE32(in := MNG_Raw32BitImage);
                        toServer.Header.Counter      := Counter;

                        toServer.Payload[1] := HOST_TO_BE32(3); (* number of signals *)

                        (* FLOAT32 Disc_00_ACT_POS *)
                        MEMCPY(destAddr := ADR(DWordBuffer), srcAddr := ADR(Outputs.Disc_00_ACT_POS), n := 4);
                        toServer.Payload[2] := HOST_TO_BE32(DWordBuffer);

                        (* FLOAT32 A2014_09_12_Left_Predeterminado_00_ACT_POS *)
                        MEMCPY(destAddr := ADR(DWordBuffer), srcAddr := ADR(Outputs.A2014_09_12_Left_Predeterminado_00_ACT_POS), n := 4);
                        toServer.Payload[3] := HOST_TO_BE32(DWordBuffer);

                        (* FLOAT32 A2014_09_12_Right_Predeterminado_00_ACT_POS *)
                        MEMCPY(destAddr := ADR(DWordBuffer), srcAddr := ADR(Outputs.A2014_09_12_Right_Predeterminado_00_ACT_POS), n := 4);
                        toServer.Payload[4] := HOST_TO_BE32(DWordBuffer);

                        toServer.Header.SentTime := HOST_TO_BE32(in := clock.systemTime.wMilliseconds + clock.systemTime.wMinute * 60000);

                        (* send frame *)
                        fbSend(bExecute  := FALSE);
                        fbSend(sSrvNetID := '',
                               hSocket   := fbConnect.hSocket,
                               cbLen     := SIZEOF(toServer.Header) + _byteCount,(* size of header + size of user data *)
                               pSrc      := ADR(toServer),(* pointer to the frame data *)
                               bExecute  := TRUE,
                               tTimeout  := T#5s);

                        tx_state := 1;
                    END_IF
                1:(* wait until send not busy *)
                    fbSend( bExecute := FALSE );
                    IF NOT fbSend.bBusy THEN
                        tx_state := 0;
                        IF NOT fbSend.bError THEN(* no error *)
                            ;
                        ELSE(* send error => log error and disconnect *)
                            errors.Error(nErrId := fbSend.nErrId );
                            bDisconnect := TRUE;(* set flag *)
                        END_IF
                    END_IF
            END_CASE

            (* ------------------------------------------- Get/fetch rx data ----------------------------------------------------------------- *)
            CASE rx_state OF
                0:
                    IF NOT bDisconnect THEN
                        pollTimer( IN := TRUE );
                        IF pollTimer.Q THEN
                            pollTimer( IN := FALSE );

                            fbReceive( bExecute := FALSE );
                            fbReceive( 	sSrvNetId	:= '',
                            hSocket		:= fbConnect.hSocket,
                            cbLen		:= SIZEOF(fromServer) - cbReceived,
                            pDest		:= ADR(fromServer) + cbReceived,
                            bExecute	:= TRUE,
                            tTimeout	:= T#5s );
                            rx_state := 1;
                        END_IF
                    END_IF
                1:(* wait until receive not busy *)
                    fbReceive( bExecute := FALSE );
                    IF NOT fbReceive.bBusy THEN
                        rx_state := 0;
                        IF NOT fbReceive.bError THEN
                            IF fbReceive.nRecBytes > 0 THEN (* some bytes received *)

                                pollTimer( PT := T#0s );(* increase polling speed *)
                                cbReceived := cbReceived + fbReceive.nRecBytes;

                                (* parse received bytes *)
                                REPEAT
                                    bAbort := TRUE;(* set flag *)
                                    IF cbReceived >= SIZEOF(fromServer.Header) THEN (* all header bytes received => check header data *)

                                        (* correct header data *)
                                        fromServer.Header.ByteCount    := BE32_TO_HOST(fromServer.Header.ByteCount);
                                        Counter                        := fromServer.Header.Counter;
                                        fromServer.Header.SentTime     := BE32_TO_HOST(fromServer.Header.SentTime);
                                        fromServer.Header.DatagramType := BE32_TO_HOST(fromServer.Header.DatagramType);

                                        IF (fromServer.Header.ByteCount <= SIZEOF( fromServer.Payload))(* check frame (user data) length *)
                                        THEN

                                            cbRx := SIZEOF(fromServer.Header) + fromServer.Header.ByteCount;(* calculate the (expected) length of the rx frame *)
                                            IF cbReceived >= cbRx  THEN (* all frame bytes received? *)

                                               (* currently only use the data on a 32 Bit raw image *)
                                                IF fromServer.Header.DatagramType = MNG_Raw32BitImage THEN

                                                    IF 20 = (fromServer.Header.ByteCount - 4) THEN

                                                        (* BOOL HallSensor1_00_IR *)
                                                        Inputs.HallSensor1_00_IR := fromServer.Payload[2]<>0;

                                                        (* BOOL HallSensor2_00_IR *)
                                                        Inputs.HallSensor2_00_IR := fromServer.Payload[3]<>0;

                                                        (* BOOL init_sensor_cookie_module_00_IR *)
                                                        Inputs.init_sensor_cookie_module_00_IR := fromServer.Payload[4]<>0;

                                                        (* BOOL kein_cookie_mehr_00_IR *)
                                                        Inputs.kein_cookie_mehr_00_IR := fromServer.Payload[5]<>0;

                                                        (* BOOL cookiebox_sensor_00_IR *)
                                                        Inputs.cookiebox_sensor_00_IR := fromServer.Payload[6]<>0;

                                                    ELSE(* receive error: invalid frame format/data *)
                                                        errors.Error(nErrId := PLCPRJ_ERROR_INVALID_IO_FORMAT_RECEIVED );
                                                    END_IF

                                                END_IF

                                                MEMMOVE( ADR( fromServer ), ADR( fromServer ) + cbRx,  cbReceived - cbRx );(* shift the remaining rx bytes *)
                                                cbReceived := cbReceived - cbRx;(* recalculate the size of the remaining rx bytes *)

                                                bAbort := FALSE;(* reset flag, try to parse next frame *)

                                                (* ELSE repeat reading *)
                                            END_IF

                                        ELSE(* receive error: invalid frame format/data *)
                                            errors.Error(nErrId := PLCPRJ_ERROR_INVALID_FRAME_FORMAT );
                                            bDisconnect := TRUE;(* set flag *)
                                        END_IF
                                        (* ELSE repeat reading *)
                                    END_IF (* IF cbReceived >= SIZEOF(rxFrame.head) THEN *)

                                UNTIL bAbort
                                END_REPEAT

                            ELSE(* fbReceive.nRecBytes = 0, repeat reading *)
                                pollTimer( PT := PLCPRJ_RECEIVER_POLLING_CYCLE_TIME );(* slow down the polling cycle *)
                            END_IF(* IF fbReceive.nRecBytes > 0 THEN *)
                        ELSE(* receive error => log error and disconnect *)
                            errors.Error(nErrId := fbReceive.nErrId );
                            bDisconnect := TRUE;(* set flag *)
                        END_IF

                    END_IF(*IF NOT fbReceive.bBusy THEN*)

            END_CASE

        END_IF

    3:(* disconnect *)
        fbConnect( bEnable:= FALSE, eState=>eState );
        IF eState = eSOCKET_DISCONNECTED THEN
            state := 0;
        END_IF

END_CASE

END_FUNCTION_BLOCK

// ---- POUs/FB_LogFifo.TcPOU
(* Log/debug/error message fifo *)
FUNCTION_BLOCK FB_LogFifo
VAR_INPUT
	bLog		: BOOL 		:= FALSE;(* TRUE => Enable log message output, FALSE => Disable *)
	sPrefix		: STRING 	:= 'Unknown::';(* Log message description string (allows the identification of log message source) *)
	
	sMessage	: STRING 	:= '';(* String message to add (write) to the fifo *)
	nErrID		: UDINT 	:= 0;(* Error code to add (write) to the fifo *)
	hSocket		: T_HSOCKET;(* Socket connection handle *)
END_VAR
VAR_OUTPUT
	bOk			: BOOL;(* TRUE = New entry added or removed succesfully, FALSE = Fifo overflow or fifo empty *)
	sGet		: T_MaxString := '';(* String entry removed (read) from fifo *)
	nCount		: UDINT := 0;(* Number of fifo entries *)
END_VAR
VAR
	fbBuffer 	: FB_StringRingBuffer;(* Basic (lower level) string buffer control function block *)
	buffer		: ARRAY[0..PLCPRJ_BUFFER_SIZE] OF BYTE;(* Internal buffer memory *)
	sSource		: T_MaxString;	
	sPut		: T_MaxString;
END_VAR

;

ACTION Remove:
(* Removes oldest fifo entry *)
IF nCount = 0 THEN
	sGet := '';
	bOk := FALSE;
	RETURN;
END_IF

fbBuffer.A_RemoveHead( pBuffer:= ADR(buffer), cbBuffer:= SIZEOF(buffer),
						getValue=>sGet, bOk=>bOk, nCount=>nCount );
END_ACTION

ACTION Clear:
(* Clears all fifo entries *)
fbBuffer.A_Reset( 	pBuffer := ADR( buffer ), cbBuffer := SIZEOF( buffer ), 
					bOk=>bOk, nCount=>nCount, getValue=>sGet );
END_ACTION

ACTION Message:
(* Adds new fifo entry *)
sPut := CONCAT( CONCAT( sPrefix, sMessage ), CONCAT( '::', HSOCKET_TO_STRING(hSocket) ) );
fbBuffer.A_AddTail( pBuffer:= ADR(buffer), cbBuffer:= SIZEOF(buffer),
					putValue:= sPut, bOk=>bOk, nCount=>nCount );
IF bOk THEN
	IF bLog THEN(* Log information message *)
		ADSLOGSTR( ADSLOG_MSGTYPE_HINT OR ADSLOG_MSGTYPE_LOG, '%s', sPut );	
	END_IF
END_IF
END_ACTION

ACTION Error:
(* Adds new fifo entry *)
IF nErrID = 0 THEN
	sSource := '::Error: 0x';
ELSIF ( nErrID AND 16#80000000) = 16#80000000 THEN
	IF nErrID = 16#80072746 THEN
		sSource := '::Win32 error (the connection is reset by remote side): 0x';
	ELSE
		sSource := '::Win32 error: 0x';
	END_IF
ELSIF (nErrID AND 16#00008100) = 16#00008100 THEN
	CASE nErrID OF
		PLCPRJ_ERROR_RECEIVE_TIMEOUT:
			sSource := '::PLC sample project receive timeout error: 0x';
		PLCPRJ_ERROR_SENDFIFO_OVERFLOW:
			sSource := '::PLC sample project send fifo overflow error: 0x';
		PLCPRJ_ERROR_RECFIFO_OVERFLOW:
			sSource := '::PLC sample project receive fifo overflow error: 0x';
		PLCPRJ_ERROR_INVALID_FRAME_FORMAT:
			sSource := '::PLC sample project invalid frame format error: 0x';
	ELSE
		sSource := '::Other PLC sample project error: 0x';
	END_CASE
ELSIF (nErrID AND 16#00008000) = 16#00008000 THEN
	sSource := '::Internal TCP/IP Connection Server error: 0x';
ELSE
	sSource := '::TwinCAT System error: 0x';
END_IF

sPut := CONCAT( CONCAT( CONCAT( sPrefix, sMessage ), sSource ), DWORD_TO_HEXSTR( nErrID AND 16#FFFF, 0, FALSE ) ); 

fbBuffer.A_AddTail( pBuffer:= ADR(buffer), cbBuffer:= SIZEOF(buffer),
					putValue:= sPut, bOk=>bOk, nCount=>nCount );
IF bOk THEN
	IF bLog THEN(* Log error message *)
		ADSLOGSTR( ADSLOG_MSGTYPE_ERROR OR ADSLOG_MSGTYPE_LOG, '%s', sPut );	
	END_IF
END_IF
END_ACTION

END_FUNCTION_BLOCK
